PROGRAM Slit_Prog
VAR
    mySlits : FB_SlitPairV2;
END_VAR

mySlits(nIdPositiveAxis:=1,nIdNegativeAxis:=2,nIdGapSizeAxis:=3,nIdGapCentreAxis:=4,bEnable:= TRUE);

END_PROGRAM

(* stored: Version 1.1.0.1, ProductVersion 3.1.4024.11
   POU Slit_Prog: Id {c85adad8-3e0e-4939-ab93-f86e8caa7aa1}, SpecialFunc None *)
